SUBAPPLICATION SIN_TO_PCAN_Callback_DWord (* Sinus-Signalgenerator (GEN_SIN) als PCAN-Callback-CAN-Botschaft senden, Wert als volle DWORD-Genauigkeit gepackt. Diagnose/Debug-Baustein zum Plotten auf PCAN Explorer. *)
  (* Standard: 61499-2 *)
  (* Version 1.0, 2026-09-09, Franz Höpfinger, Meisterschulen am Ostbahnhof, Ausgelagert aus Uebung_126b2_sub zur Wiederverwendung. *)
  PACKAGE MyLib::sys;
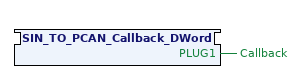
  PLUGS
    PLUG1 : isobus::pgn::tx::Callback;
  END_PLUGS
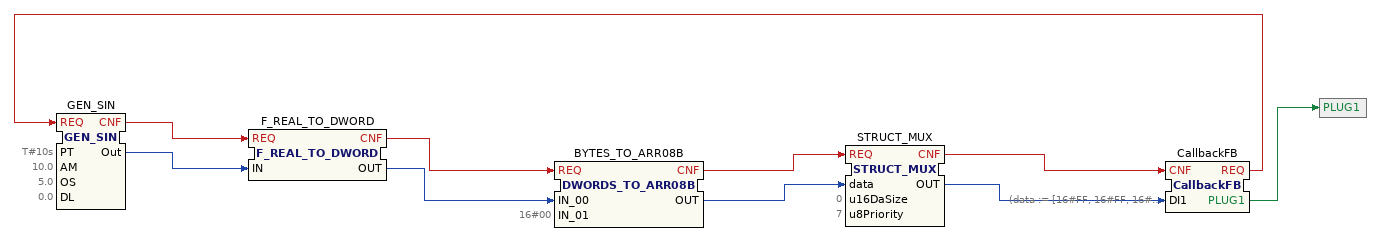
  FBS
    CallbackFB : isobus::pgn::tx::CallbackFB(DI1 := (data := [16#FF, 16#FF, 16#FF, 16#FF, 16#FF, 16#FF, 16#FF, 16#FF]));
    STRUCT_MUX : eclipse4diac::convert::STRUCT_MUX(u16DaSize := 0, u8Priority := 7); {SET_ATTRIBUTE(StructuredType, isobus::pgn::CAN_MSG)}
    BYTES_TO_ARR08B : logiBUS::utils::conversion::arr::reversing::DWORDS_TO_ARR08B(IN_01 := 16#00);
    GEN_SIN : OSCAT::Basic::POUs::Engineering::signal_generators::GEN_SIN(PT := T#10s, AM := 10.0, OS := 5.0, DL := 0.0);
    F_REAL_TO_DWORD : iec61131::conversion::F_REAL_TO_DWORD;
  END_FBS
  EVENT_CONNECTIONS
    STRUCT_MUX.CNF TO CallbackFB.CNF;
    BYTES_TO_ARR08B.CNF TO STRUCT_MUX.REQ;
    CallbackFB.REQ TO GEN_SIN.REQ;
    GEN_SIN.CNF TO F_REAL_TO_DWORD.REQ;
    F_REAL_TO_DWORD.CNF TO BYTES_TO_ARR08B.REQ;
  END_CONNECTIONS
  DATA_CONNECTIONS
    STRUCT_MUX.OUT TO CallbackFB.DI1;
    BYTES_TO_ARR08B.OUT TO STRUCT_MUX.data;
    GEN_SIN.Out TO F_REAL_TO_DWORD.IN;
    F_REAL_TO_DWORD.OUT TO BYTES_TO_ARR08B.IN_00;
  END_CONNECTIONS
  ADAPTER_CONNECTIONS
    CallbackFB.PLUG1 TO PLUG1;
  END_CONNECTIONS
END_SUBAPPLICATION
